Universal Robots PolyScope program: yol1pr.urp

Program yol1pr (installation=default directory=/programs createdIn=5.14.5 lastSavedIn=5.14.5 robotSerialNumber=20195300809)
Calibrated DH parameters: a=[-0.000085, -0.20076, -0.212369, 0.000121, -0.000118, 0]; d=[0.15185, -26.306375, 24.753047, 1.684739, 0.085386, 0.092088]; alpha=[1.572149, -0.00522, -0.011864, 1.571339, -1.571085, 0]; deltaTheta=[0, 0.599885, -0.513355, -0.086555, 0.000006, 0]
InitVariablesNode
BeforeStart
  var_1 := socket_open("10.5.20.90",29999)
  Loop While (checkContinuously=false) expression=var_1≟ False
    var_1 := socket_open("10.5.20.90",29999)
Robot Program (runOnlyOnce=false)
  Popup Message (haltProgram=false message=hola matlab inputType=Text)
